% RSLogix 500 project compare Question 1 to 5.RSS, saved by version 8.30.00.15 %
PROJECT "UNTITLED"    % processor: MicroLogix 1000 %

PROGRAM FILES
  LAD 2 "MAIN_PROG"  7 rungs
  LAD 3 "USER_FAULT"  1 rungs
  LAD 4 "HSC_INT"  1 rungs
  LAD 5 "STI_INT"  1 rungs
  LAD 6, 7, 8, 9, 10, 11, 12, 13, 14, 15, 16: only END

DATA FILES
  O0 OUTPUT  1 elements
  I1 INPUT  2 elements
  S2 STATUS  33 elements
  B3 BINARY  32 elements
  T4 TIMER  40 elements
  C5 COUNTER  32 elements
  R6 CONTROL  16 elements
  N7 INTEGER  105 elements

LADDER 2 "MAIN_PROG"
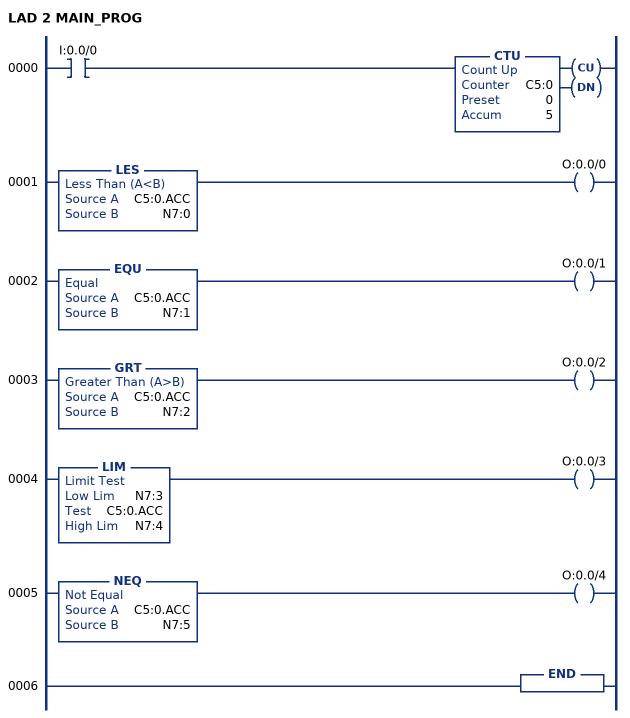
% Rung: 0 %
SOR XIC I:0.0/0 CTU C5:0 0 5 EOR
% Rung: 1 %
SOR LES C5:0.ACC N7:0 OTE O:0.0/0 EOR
% Rung: 2 %
SOR EQU C5:0.ACC N7:1 OTE O:0.0/1 EOR
% Rung: 3 %
SOR GRT C5:0.ACC N7:2 OTE O:0.0/2 EOR
% Rung: 4 %
SOR LIM N7:3 C5:0.ACC N7:4 OTE O:0.0/3 EOR
% Rung: 5 %
SOR NEQ C5:0.ACC N7:5 OTE O:0.0/4 EOR
% Rung: 6 %
SOR END EOR

DATA TABLE (non-zero values as saved)
DATA C5
% .PRE .ACC %
% C5:0 % 0 5
DATA N7
% N7:0 % 4 4 4 3 6 4 0 0 0 0
